TYPE ST_System_WDT_Stellwert :
STRUCT
	Anford_Stellventil_Netz				: BOOL;
	Anford_Pumpe_Netz					: BOOL;
	Anford_Stellventil					: BOOL;
	Anford_Pumpe						: BOOL;
	Anford_Regelventil					: BOOL;
	Anford_Aussenfassadenaktivierung	: BOOL;

	Temp_Vorl							: REAL;
END_STRUCT
END_TYPE

(* stored: Version 1.1.0.1, ProductVersion 3.1.4024.9
   DUT ST_System_WDT_Stellwert: Id {c8f2e438-3d03-4939-9bad-383dcea62bb8} *)
